TYPE Type_ModuleCommIn_Test :
STRUCT
	m_Work					:BOOL;
	m_OutOfArea				:BOOL;
	m_PartDropped			:BOOL;
END_STRUCT
END_TYPE

(* stored: Version 1.1.0.1, ProductVersion 3.1.4024.3
   DUT Type_ModuleCommIn_Test: Id {8fbbd775-a49e-44aa-8b85-4001f591fc05} *)
